# EPICS autosave request: measComp/measCompApp/Db/measCompAnalogOut_settings.req
$(P)$(R)Pulse
$(P)$(R)TweakVal
